{attribute 'qualified_only'}
{attribute 'strict'}
TYPE ESpecialAlarmIds :
(
	none := 0,
	recovery_request := 990,
	definition_request := 991
) UINT;
END_TYPE

(* stored: Version 1.1.0.1, ProductVersion 3.1.4024.9
   DUT ESpecialAlarmIds: Id {280426ea-874f-4891-8547-bd46f7a3a383} *)
